FUNCTION_BLOCK FB4
VAR_INPUT
	fbGenericFB : iFb;
	fInput1: REAL;
	fInput2: REAL; 
END_VAR
VAR_OUTPUT
	bIsEven : BOOL;
END_VAR
VAR
	iResult : INT;
END_VAR


//Inizializzo e uso la FB Generica grazie all'interfaccia
fbGenericFB.fInput1 := fInput1;
fbGenericFB.fInput2 := fInput2;

iResult := REAL_TO_INT(fbGenericFB.returnValue());

//Calcolo l'output
bIsEven := (iResult MOD 2) = 0;

END_FUNCTION_BLOCK

(* stored: Version 1.1.0.1, ProductVersion 3.1.4022.16
   POU FB4: Id {6f088c33-22ac-4c78-869b-1f3b9b7ebff3}, SpecialFunc None *)
